Staubli VAL3: interfaceCS8.pjx

--- interfaceCS8.pjx ---
Parameters version=s7.11 stackSize=5000 millimeterUnit=true
Program file=ack.pgx
Program file=clearScreen.pgx
Program file=debug.pgx
Program file=feedbackStatus.pgx
Program file=init.pgx
Program file=motionBuffer.pgx
Program file=motionProgress.pgx
Program file=motionStatus.pgx
Program file=start.pgx
Program file=stop.pgx
Program file=trajBuffer.pgx
Program file=velOverwrite.pgx
Data file=interfaceCS8.dtx
Library alias=libQueueFuncs path=Disk://ros_libs/QueueFuncs/QueueFuncs.pjx

--- interfaceCS8.dtx ---
mdesc mNomSpeed
screen scMonitor

--- start.pgx ---
program start()
begin

  // Library to handle all of the interface actions for CS8 controller
  // Loaded at runtime in ros_server()

  // DO NOT auto-load
  // Auto-loading will break cross-controller functionality
  // The correct library will be loaded at runtime, otherwise an error will be generated

end

--- ack.pgx ---
public program ack(num x_nHeaderTime, num x_nElapsedTime)
begin

  gotoxy(scMonitor, 0,9)
  put(scMonitor, "recvMsgHeader:")
  gotoxy(scMonitor, 15,9)
  put(scMonitor, toString(".4", x_nHeaderTime))

  gotoxy(scMonitor, 0,10)
  put(scMonitor, "other states:")
  gotoxy(scMonitor, 15,10)
  put(scMonitor, toString(".4", x_nElapsedTime))

end

--- clearScreen.pgx ---
public program clearScreen()
begin

  cls(scMonitor)

end

--- debug.pgx ---
public program debug(num& x_nExecStatus)
begin

  gotoxy(scMonitor, 18,12)
  switch x_nExecStatus
    case 0
      put(scMonitor, "[+]")
      x_nExecStatus = 1
    break
    case 1
      put(scMonitor, "[-]")
      x_nExecStatus = 0
    break
    default
    break
  endSwitch

end

--- feedbackStatus.pgx ---
public program feedbackStatus(num x_nOutConnFlag)
begin

  // update connection status on port 11002
  gotoxy(scMonitor, 0,1)
  // 11 characteres: gotoxy(12,1) to insert status
  put(scMonitor, "Port 11002:")
  gotoxy(scMonitor, 12,1)
  switch x_nOutConnFlag
    case -1
      put(scMonitor, "connection lost")
    break
    case 0
      put(scMonitor, "not connected")
    break
    case 1
      put(scMonitor, "connected")
    break
    default
      put(scMonitor, "not connected")
    break
  endSwitch

end

--- init.pgx ---
public program init()
begin


  userPage(scMonitor)
  cls(scMonitor)
  title(scMonitor, "ROS-I server")

end

--- motionBuffer.pgx ---
public program motionBuffer(num x_nMovePts, num x_nElems)
begin

  gotoxy(scMonitor, 0,4)
  put(scMonitor, "Motion buffer:")
  gotoxy(scMonitor, 19,4)
  put(scMonitor, x_nElems)
  gotoxy(scMonitor, 24,4)
  put(scMonitor, x_nMovePts)

end

--- motionProgress.pgx ---
public program motionProgress(num x_nMoveId, num x_nMotProg)
begin

  gotoxy(scMonitor, 0,7)
  put(scMonitor, "moveId:")
  gotoxy(scMonitor, 8,7)
  put(scMonitor, x_nMoveId)
  gotoxy(scMonitor, 13,7)
  put(scMonitor, "progress:")
  gotoxy(scMonitor, 23,7)
  put(scMonitor, x_nMotProg)

end

--- motionStatus.pgx ---
public program motionStatus(num x_nInConnFlag)
begin

  // update connection status on port 11000
    gotoxy(scMonitor, 0,0)
    // 11 characteres: gotoxy(12,0) to insert status
    put(scMonitor, "Port 11000:")
    gotoxy(scMonitor, 12,0)
    switch x_nInConnFlag
      case -1
        put(scMonitor, "connection lost")
      break
      case 0
        put(scMonitor, "not connected")
      break
      case 1
        put(scMonitor, "connected")
      break
      default
        put(scMonitor, "not connected")
      break
    endSwitch

end

--- trajBuffer.pgx ---
public program trajBuffer(num x_nElems, num x_nPtsPopped)
begin

  gotoxy(scMonitor, 0,3)
  // 18 characteres: gotoxy(19,3) to insert status
  put(scMonitor, "Trajectory buffer:")
  gotoxy(scMonitor, 19,3)
  put(scMonitor, x_nElems)
  // also print number of points popped from buffer
  gotoxy(scMonitor, 24,3)
  put(scMonitor, x_nPtsPopped)

end

--- velOverwrite.pgx ---
public program velOverwrite(bool x_bOverwriteVel)
begin

  gotoxy(scMonitor, 0,5)
  put(scMonitor, "Velocity overwrite:")
  gotoxy(scMonitor, 20,5)
  if(x_bOverwriteVel == true)
    put(scMonitor, "enabled")
  else
    put(scMonitor, "disabled")
  endIf

end
